# EPICS SNL sequencer program: ioc/etheripIOCApp/src/sncSabia.stt
program sncSabia

%%//----------------------------------------
%%//    Global Variables
%%//----------------------------------------

%%//----------------------------------------
%%//    Monitored PVs - High Level
%%//----------------------------------------

int pos_tolerance_sp;
assign pos_tolerance_sp to "{P}{R}PosTolerance-SP";
monitor pos_tolerance_sp;

int change_pol_evt;
assign change_pol_evt to "{P}{R}ChangePolFlg";
monitor change_pol_evt;
evflag change_pol_evt_flg;
sync change_pol_evt change_pol_evt_flg;

int pol_type_sel;
assign pol_type_sel to "{P}{R}PolType-Sel";
monitor pol_type_sel;
evflag pol_type_sel_flg;
sync pol_type_sel pol_type_sel_flg;

int change_gain_evt;
assign change_gain_evt to "{P}{R}ChangeGainFlg";
monitor change_gain_evt;
evflag change_gain_evt_flg;
sync change_gain_evt change_gain_evt_flg;

int gain_motion_type_sel;
assign gain_motion_type_sel to "{P}{R}GainMotionType-Sel";
monitor gain_motion_type_sel;
evflag gain_motion_type_sel_flg;
sync gain_motion_type_sel gain_motion_type_sel_flg;

int energy_sp;
assign energy_sp to "{P}{R}Energy-SP";
monitor energy_sp;
evflag energy_sp_flg;
sync energy_sp energy_sp_flg;

int k_sp;
assign k_sp to "{P}{R}K-SP";
monitor k_sp;
evflag k_sp_flg;
sync k_sp k_sp_flg;

int shift_sp;
assign shift_sp to "{P}{R}Shift-SP";
monitor shift_sp;
evflag shift_sp_flg;
sync shift_sp shift_sp_flg;

int start_escan_evt;
assign start_escan_evt to "{P}{R}StartEScanFlg";
monitor start_escan_evt;
evflag start_escan_evt_flg;
sync start_escan_evt start_escan_evt_flg;

int escan_start_pos_sp;
assign escan_start_pos_sp to "{P}{R}EScanStartPos-SP";
monitor escan_start_pos_sp;
evflag escan_start_pos_sp_flg;
sync escan_start_pos_sp escan_start_pos_sp_flg;

int escan_end_pos_sp;
assign escan_end_pos_sp to "{P}{R}EScanEndPos-SP";
monitor escan_end_pos_sp;
evflag escan_end_pos_sp_flg;
sync escan_end_pos_sp escan_end_pos_sp_flg;

int pol_mode_velo_sp;
assign pol_mode_velo_sp to "{P}{R}PolModeVelo-SP";
monitor pol_mode_velo_sp;
evflag pol_mode_velo_sp_flg;
sync pol_mode_velo_sp pol_mode_velo_sp_flg;

int pol_mode_acc_sp;
assign pol_mode_acc_sp to "{P}{R}PolModeAcc-SP";
monitor pol_mode_acc_sp;
evflag pol_mode_acc_sp_flg;
sync pol_mode_acc_sp pol_mode_acc_sp_flg;

int energy_mode_velo_sp;
assign energy_mode_velo_sp to "{P}{R}EnergyModeVelo-SP";
monitor energy_mode_velo_sp;
evflag energy_mode_velo_sp_flg;
sync energy_mode_velo_sp energy_mode_velo_sp_flg;

int energy_mode_acc_sp;
assign energy_mode_acc_sp to "{P}{R}EnergyModeAcc-SP";
monitor energy_mode_acc_sp;
evflag energy_mode_acc_sp_flg;
sync energy_mode_acc_sp energy_mode_acc_sp_flg;

int max_velo_sp;
assign max_velo_sp to "{P}{R}MaxVelo-SP";
monitor max_velo_sp;
evflag max_velo_sp_flg;
sync max_velo_sp max_velo_sp_flg;

int max_acc_sp;
assign max_acc_sp to "{P}{R}MaxAcc-SP";
monitor max_acc_sp;
evflag max_acc_sp_flg;
sync max_acc_sp max_acc_sp_flg;

int parking_request_evt;
assign parking_request_evt to "{P}{R}ParkingRequestFlg";
monitor parking_request_evt;
evflag parking_request_evt_flg;
sync parking_request_evt parking_request_evt_flg;

int parking_pol_sp;
assign parking_pol_sp to "{P}{R}ParkingPol-SP";
monitor parking_pol_sp;
evflag parking_pol_sp_flg;
sync parking_pol_sp parking_pol_sp_flg;

int parking_energy_sp;
assign parking_energy_sp to "{P}{R}ParkingEnergy-SP";
monitor parking_energy_sp;
evflag parking_energy_sp_flg;
sync parking_energy_sp parking_energy_sp_flg;

int get_parking_request_evt;
assign get_parking_request_evt to "{P}{R}GetParkingRequestFlg";
monitor get_parking_request_evt;
evflag get_parking_request_evt_flg;
sync get_parking_request_evt get_parking_request_evt_flg;

int actual_pol_displacement_mon;
assign actual_pol_displacement_mon to "{P}{R}ActualPolDisplacement-Mon";
monitor actual_pol_displacement_mon;

int actual_pol_mon;
assign actual_pol_mon to "{P}{R}ActualPol-Mon";
monitor actual_pol_mon;

int actual_k_displacement_mon;
assign actual_k_displacement_mon to "{P}{R}ActualKDisplacement-Mon";
monitor actual_k_displacement_mon;

int actual_k_mon;
assign actual_k_mon to "{P}{R}ActualK-Mon";
monitor actual_k_mon;

int actual_energy_mon;
assign actual_energy_mon to "{P}{R}ActualEnergy-Mon";
monitor actual_energy_mon;

%%// Conversion Coefficients - Shift to K

int conv_shift_to_k_a0_sp;
assign conv_shift_to_k_a0_sp to "{P}{R}ConvShiftToKA0-SP";
monitor conv_shift_to_k_a0_sp;

int conv_shift_to_k_a1_sp;
assign conv_shift_to_k_a1_sp to "{P}{R}ConvShiftToKA1-SP";
monitor conv_shift_to_k_a1_sp;

int conv_shift_to_k_a2_sp;
assign conv_shift_to_k_a2_sp to "{P}{R}ConvShiftToKA2-SP";
monitor conv_shift_to_k_a2_sp;

int conv_shift_to_k_a3_sp;
assign conv_shift_to_k_a3_sp to "{P}{R}ConvShiftToKA3-SP";
monitor conv_shift_to_k_a3_sp;

int conv_shift_to_k_a4_sp;
assign conv_shift_to_k_a4_sp to "{P}{R}ConvShiftToKA4-SP";
monitor conv_shift_to_k_a4_sp;

int conv_shift_to_k_a5_sp;
assign conv_shift_to_k_a5_sp to "{P}{R}ConvShiftToKA5-SP";
monitor conv_shift_to_k_a5_sp;

int conv_shift_to_k_a6_sp;
assign conv_shift_to_k_a6_sp to "{P}{R}ConvShiftToKA6-SP";
monitor conv_shift_to_k_a6_sp;

int conv_shift_to_k_a7_sp;
assign conv_shift_to_k_a7_sp to "{P}{R}ConvShiftToKA7-SP";
monitor conv_shift_to_k_a7_sp;

int conv_shift_to_k_a8_sp;
assign conv_shift_to_k_a8_sp to "{P}{R}ConvShiftToKA8-SP";
monitor conv_shift_to_k_a8_sp;

%%// Conversion Coefficients - K to Energy

int conv_k_to_energy_a0_sp;
assign conv_k_to_energy_a0_sp to "{P}{R}ConvKToEnergyA0-SP";
monitor conv_k_to_energy_a0_sp;

int conv_k_to_energy_a1_sp;
assign conv_k_to_energy_a1_sp to "{P}{R}ConvKToEnergyA1-SP";
monitor conv_k_to_energy_a1_sp;

int conv_k_to_energy_a2_sp;
assign conv_k_to_energy_a2_sp to "{P}{R}ConvKToEnergyA2-SP";
monitor conv_k_to_energy_a2_sp;

int conv_k_to_energy_a3_sp;
assign conv_k_to_energy_a3_sp to "{P}{R}ConvKToEnergyA3-SP";
monitor conv_k_to_energy_a3_sp;

int conv_k_to_energy_a4_sp;
assign conv_k_to_energy_a4_sp to "{P}{R}ConvKToEnergyA4-SP";
monitor conv_k_to_energy_a4_sp;

int conv_k_to_energy_a5_sp;
assign conv_k_to_energy_a5_sp to "{P}{R}ConvKToEnergyA5-SP";
monitor conv_k_to_energy_a5_sp;

int conv_k_to_energy_a6_sp;
assign conv_k_to_energy_a6_sp to "{P}{R}ConvKToEnergyA6-SP";
monitor conv_k_to_energy_a6_sp;

int conv_k_to_energy_a7_sp;
assign conv_k_to_energy_a7_sp to "{P}{R}ConvKToEnergyA7-SP";
monitor conv_k_to_energy_a7_sp;

int conv_k_to_energy_a8_sp;
assign conv_k_to_energy_a8_sp to "{P}{R}ConvKToEnergyA8-SP";
monitor conv_k_to_energy_a8_sp;

%%//----------------------------------------
%%//    Output PVs - High Level
%%//----------------------------------------

int enbl_low_lvl_ctrl_proc;
assign enbl_low_lvl_ctrl_proc to "{P}{R}EnblLowLvlCtrl.PROC";

int dsbl_low_lvl_ctrl_proc;
assign dsbl_low_lvl_ctrl_proc to "{P}{R}DsblLowLvlCtrl.PROC";

%%//----------------------------------------
%%//    Monitored PVs - Low Level
%%//----------------------------------------

int mod_01_motion_state_mon;
assign mod_01_motion_state_mon to "{P}{R}Mod01MotionState-Mon";
monitor mod_01_motion_state_mon;

%%//----------------------------------------
%%//    Output PVs - Low Level
%%//----------------------------------------

int mod_01_rel_pos_sp;
assign mod_01_rel_pos_sp to "{P}{R}Mod01RelPos-SP";

int mod_01_velo_sp;
assign mod_01_velo_sp to "{P}{R}Mod01Velo-SP";

int mod_01_acc_sp;
assign mod_01_acc_sp to "{P}{R}Mod01Acc-SP";

int mod_01_decel_sp;
assign mod_01_decel_sp to "{P}{R}Mod01Decel-SP";

int mod_01_phy_cid_actual_pos_mon;
assign mod_01_phy_cid_actual_pos_mon to "{P}{R}Mod01PhyCIDActualPos-Mon";

int mod_01_phy_cie_actual_pos_mon;
assign mod_01_phy_cie_actual_pos_mon to "{P}{R}Mod01PhyCIEActualPos-Mon";

int mod_01_phy_csd_actual_pos_mon;
assign mod_01_phy_csd_actual_pos_mon to "{P}{R}Mod01PhyCSDActualPos-Mon";

int mod_01_phy_cse_actual_pos_mon;
assign mod_01_phy_cse_actual_pos_mon to "{P}{R}Mod01PhyCSEActualPos-Mon";

int mod_01_coup_sel;
assign mod_01_coup_sel to "{P}{R}Mod01Coup-Sel";

int mod_01_trig_type_sel;
assign mod_01_trig_type_sel to "{P}{R}Mod01TrigType-Sel";

int mod_01_ref_type_sel;
assign mod_01_ref_type_sel to "{P}{R}Mod01RefType-Sel";

int inter_mod_coup_sel;
assign inter_mod_coup_sel to "{P}{R}InterModCoup-Sel";

int mod_01_mirror_sel;
assign mod_01_mirror_sel to "{P}{R}Mod01Mirror-Sel";

int mod_01_soft_trig_cmd;
assign mod_01_soft_trig_cmd to "{P}{R}Mod01SoftTrig-Cmd";

%%//----------------------------------------
%%//        Escaped C Code
%%//----------------------------------------

// required for calling seq_pvPut, seq_pvGet from embedded C code
foreign ssId;

%%#include <unistd.h>
%%#include <string.h>
%%#include "Logger.h"

// coupling modes
%%#define COUPLING_UNCOUPLED 0
%%#define COUPLING_ALL 1
%%#define COUPLING_PHASE 2
%%#define COUPLING_COUNTERPHASE 3
%%#define COUPLING_GV 4
%%#define COUPLING_GH 5

// main polarization positions (mm)
%%#define POL_LIN_VERT -26.25
%%#define POL_CIRC_RIGHT -13.125
%%#define POL_LIN_HOR 0.0
%%#define POL_CIRC_LEFT 13.125
%%// #define POL_LIN_VERT 26.25

// trigger
%%#define TRIG_TYPE_BOTH 0
%%#define TRIG_TYPE_SOFT 1
%%#define TRIG_TYPE_HARD 2

// inter-module coupling
%%#define INTER_MOD_COUPLING_001 1

// motion reference type
%%#define REFERENCE_TYPE_INTERNAL 0
%%#define REFERENCE_TYPE_EXTERNAL 1

// coupling mirror config
%%#define MIRROR_DISABLE 0
%%#define MIRROR_ENABLE 1

// motion state
%%#define MOTION_STATE_MOVING 0
%%#define MOTION_STATE_DONE 1

%%//----------------------------------------
%%//        State Notation Language
%%//----------------------------------------

ss motion_control {
    state init {
	when (delay(5.0)) {

            LOG_INFO("[%s%s] Initialization start\n", macValueGet("P"), macValueGet("R"));
	} state ready
    }

    state ready {
        entry {
            /* clear event flags to avoid
               old running invalid commands */
            efClear(change_pol_evt);
            efClear(change_gain_evt);
	    efClear(start_escan_evt);
            efClear(parking_request_evt);
            efClear(get_parking_request_evt);
        }

	when (efTestAndClear(change_pol_evt)) {
        } state change_pol

	when (efTestAndClear(change_gain_evt)) {
        } state change_gain

	when (efTestAndClear(start_escan_evt)) {
        } state start_escan

	when (efTestAndClear(parking_request_evt)) {
        } state start_parking

	when (efTestAndClear(get_parking_request_evt)) {
        } state get_parking_pos
    }

    state change_pol {

        entry {

            // local variables
            float var_target_pol, var_pos_diff;
            char var_check;

            // find target polarization
            if (pol_type_sel == 0) {
                var_target_pol = POL_CIRC_RIGHT;
            }
            else if (pol_type_sel == 1) {
                var_target_pol = POL_CIRC_LEFT;
            }
            else if (pol_type_sel == 2) {
                var_target_pol = POL_LIN_VERT;
            }
            else if (pol_type_sel == 3) {
                var_target_pol = POL_LIN_HOR;
            }

            // calculate position diff
            var_pos_diff = var_target_pol - actual_pol_displacement_mon;

            // check if diff is inside tolerance
            var_check = 1;
            if (var_pos_diff > pos_tolerance_sp
                || var_pos_diff < -pos_tolerance_sp) {

                var_check = 0;
            }

            // move to position
            if (check == 1) {
                // configure trigger to software
                mod_01_trig_type_sel = TRIG_TYPE_SOFT;
                pvPut(mod_01_trig_type_sel, SYNC);

                // make sure inter module coupling is right
                inter_mod_coup_sel = INTER_MOD_COUPLING_001;
                pvPut(inter_mod_coup_sel, SYNC);

                // configure motion reference type
                mod_01_ref_type_sel = REFERENCE_TYPE_INTERNAL;
                pvPut(mod_01_ref_type_sel, SYNC);

                // select phase coupling
                mod_01_coup_sel = COUPLING_PHASE;
                pvPut(mod_01_coup_sel, SYNC);

                // make sure mirror is disabled
                mod_01_mirror_sel = MIRROR_DISABLE;
                pvPut(mod_01_mirror_sel, SYNC);

                // configure velocity
                mod_01_velo_sp = pol_mode_velo_sp;
                pvPut(mod_01_velo_sp, SYNC);
                // configure acceleration
                mod_01_acc_sp = pol_mode_acc_sp;
                pvPut(mod_01_acc_sp, SYNC);
                // configure deceleration equal acceleration
                mod_01_decel_sp = pol_mode_acc_sp;
                pvPut(mod_01_decel_sp, SYNC);
                // configure relative position
                mod_01_rel_pos_sp = var_pos_diff;
                pvPut(mod_01_rel_pos_sp, SYNC);

                // send soft trigger to start motion
                mod_01_soft_trig_cmd = 1;
                pvPut(mod_01_soft_trig_cmd, SYNC);
            }
        }

        when (delay(1.0) && mod_01_motion_state_mon == MOTION_STATE_DONE) {
        } state ready
    }

    state change_gain {
        entry {
        }

        when (delay(1.0) && mod_01_motion_state_mon == MOTION_STATE_DONE) {
        } state ready
    }

    state start_escan {
        entry {
        }

        when (delay(1.0) && mod_01_motion_state_mon == MOTION_STATE_DONE) {
        } state ready
    }

    state start_parking {
        entry {
        }

        when (delay(1.0) && mod_01_motion_state_mon == MOTION_STATE_DONE) {
        } state ready
    }

    state get_parking_pos {
        entry {
        }

        when () {
        } state ready
    }

}
